FUNCTION_BLOCK T_RoboConnect_GetToolAnalogOutput_IncorrectIndexFails EXTENDS T_UnitTestBase
VAR
  robot : I_RoboConnect;
  targetDO : UINT;
  myTestState, prevState :
    (INIT,
    ARRANGE,
    ACT,
    ASSERT) := INIT;
  expected : BOOL;
  actual : BOOL := TRUE;
  counter : UINT;
  returnedTask : I_Task;
  resultTask : I_NumberResultTask;
END_VAR

CASE myTestState OF
  INIT:
    StateChanged();
    myTestState := ARRANGE;

  ARRANGE:
    IF StateChanged() THEN
      expected := FALSE;
      myTestState := ACT;
    END_IF

  ACT:
    actual := robot.GetToolAnalogOutput(targetDO, task => resultTask);
    myTestState := ASSERT;

  ASSERT:
    assertion.AssertEquals_BOOL(expected, actual, 'robot.GetToolAnalogOutput(targetDO, task => returnedTask)');
    TestFinished();
    myTestState := INIT;

END_CASE

METHOD FB_init : BOOL
VAR_INPUT
  bInitRetains : BOOL; // if TRUE, the retain variables are initialized (warm start / cold start)
  bInCopyCode : BOOL; // if TRUE, the instance afterwards gets moved into the copy code (online change)
  TestSuite : tcl_SimpleUnitTestLibrary.I_TestSuite;
  robot : I_TcRobot;
  targetDo : UINT;
END_VAR
THIS^.robot := robot;
THIS^.targetDo := targetDo;
END_METHOD

METHOD PRIVATE StateChanged : BOOL
IF  myTestState = prevState THEN
  RETURN;
END_IF

prevState := myTestState;
StateChanged := TRUE;
END_METHOD

METHOD WaitForCycles : BOOL
VAR_INPUT
  maxCount : UINT;
END_VAR
counter := counter + 1;

IF counter = maxCount THEN
  counter := 0;
  WaitForCycles := TRUE;
END_IF
END_METHOD

END_FUNCTION_BLOCK

(* stored: Version 1.1.0.1
   POU T_TcRobot_GetToolAnalogOutput_IncorrectIndexFails: Id {31859906-2ef8-4cc4-911b-8fe121b3afde}, SpecialFunc None
   Method FB_init: Id {7d3425d2-b20c-4163-a5f6-99c9ed52254b}
   Method StateChanged: Id {a3871735-130a-4b70-b705-be4d5d517794}
   Method WaitForCycles: Id {220dc92e-5fc6-413d-bc26-89101ecc0811} *)
